FUNCTION_BLOCK FB_SendPosVelocity
VAR_INPUT
	positionDelft : LREAL;
	VelocityDelft : LREAL;
END_VAR
VAR_OUTPUT
END_VAR
VAR
	TxMessage : EXTCANQUEUE;
	i : INT;
	Position_Values : ARRAY[0..3] OF BYTE;
	Velocity_Values : ARRAY[0..1] OF BYTE;
END_VAR
VAR_IN_OUT
	CAN_OUTPUTS : CANTXQUEUESTRUCT_E_32;
	CAN_INPUTS : CANRXQUEUESTRUCT_E_32;
END_VAR

(*
Position_Values[3] := DINT_TO_BYTE(positionDelft AND 16#FF);
Position_Values[2] := DINT_TO_BYTE(SHR(positionDelft, 8) AND 16#FF);
Position_Values[1] := DINT_TO_BYTE(SHR(positionDelft, 16) AND 16#FF);
Position_Values[0] := DINT_TO_BYTE(SHR(positionDelft, 24) AND 16#FF);

Velocity_Values[1] := DINT_TO_BYTE(VelocityDelft AND 16#FF);
Velocity_Values[0] := DINT_TO_BYTE(SHR(VelocityDelft, 8) AND 16#FF);
*)

Position_Values[3] := DINT_TO_BYTE(LREAL_TO_DINT(positionDelft*100) AND 16#FF);
Position_Values[2] := DINT_TO_BYTE(SHR(LREAL_TO_DINT(positionDelft*100), 8) AND 16#FF);
Position_Values[1] := DINT_TO_BYTE(SHR(LREAL_TO_DINT(positionDelft*100), 16) AND 16#FF);
Position_Values[0] := DINT_TO_BYTE(SHR(LREAL_TO_DINT(positionDelft*100), 24) AND 16#FF);

Velocity_Values[1] := INT_TO_BYTE(LREAL_TO_INT(VelocityDelft) AND 16#FF);
Velocity_Values[0] := INT_TO_BYTE(SHR(LREAL_TO_INT(VelocityDelft), 8) AND 16#FF);

TxMessage.cobId := 800;
TxMessage.length := 6;
FOR i := 0 TO 5 DO 
	IF i < 4 THEN 
		TxMessage.data[i] := Position_Values[i];
	ELSE 
		TxMessage.data[i] := Velocity_Values[i - 4];
	END_IF
END_FOR
CAN_OUTPUTS.TxMessages[4] := TxMessage;
//CAN_OUTPUTS.NoOfTxMessages := 1

(*
TxMessage.cobId := 800;
TxMessage.length := 6;
FOR i := 0 TO 5 DO 
	IF i < 4 THEN 
		TxMessage.data[i] := Position_Values[i];
	ELSE 
		TxMessage.data[i] := Velocity_Values[i - 4];
	END_IF
END_FOR
CAN_OUTPUTS.TxMessages[4] := TxMessage;
CAN_OUTPUTS.TxCounter := CAN_INPUTS.TxCounter + 1;
*)

END_FUNCTION_BLOCK

(* stored: Version 1.1.0.1
   POU FB_SendPosVelocity_1: Id {81cfaa36-55a9-4d26-b7b5-fec5865831f5}, SpecialFunc None *)
